// TIA Portal project "SCDW_TEST_67391275" (V17)

(* hardware
DEVICE "SCDW_TEST_PLC"  S7-1200 Station
   slot 0: "Rack_0"  S7-1200 Rack  Rack  V1.0
   slot 1: "SCDW_TEST_PLC"  CPU 1214C AC/DC/Rly  6ES7 214-1BG40-0XB0  V4.4
*)

// ===== PLC "SCDW_TEST_PLC"  CPU 1214C AC/DC/Rly =====

ORGANIZATION_BLOCK "Main"   // OB1, LAD, ProgramCycle
TITLE = "Main Program Sweep (Cycle)"
{ S7_Optimized_Access := 'TRUE' }
VERSION : 0.1
   VAR_INPUT
      Initial_Call : Bool;   // Initial call of this OB
      Remanence : Bool;   // =True, if remanent data are available
   END_VAR
BEGIN

REGION Network 1
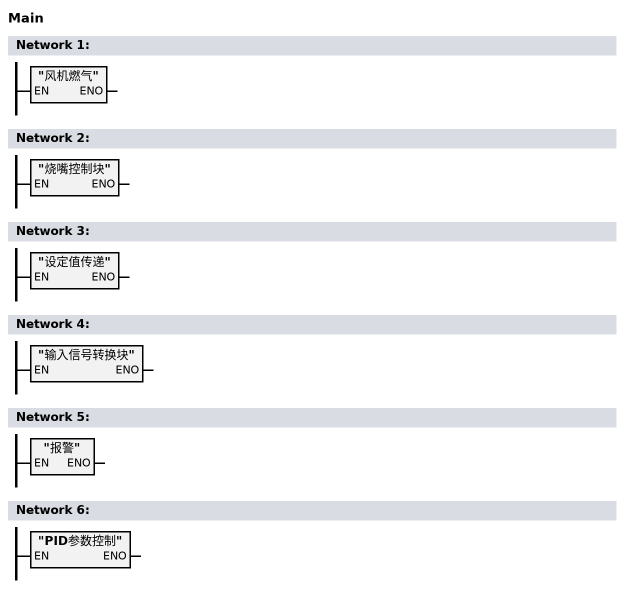
   RUNG wire#powerrail
      "风机燃气"()
   END_RUNG
   // the same network as SCL:
   "风机燃气"();
END_REGION

REGION Network 2
   RUNG wire#powerrail
      "烧嘴控制块"()
   END_RUNG
   // the same network as SCL:
   "烧嘴控制块"();
END_REGION

REGION Network 3
   RUNG wire#powerrail
      "设定值传递"()
   END_RUNG
   // the same network as SCL:
   "设定值传递"();
END_REGION

REGION Network 4
   RUNG wire#powerrail
      "输入信号转换块"()
   END_RUNG
   // the same network as SCL:
   "输入信号转换块"();
END_REGION

REGION Network 5
   RUNG wire#powerrail
      "报警"()
   END_RUNG
   // the same network as SCL:
   "报警"();
END_REGION

REGION Network 6
   RUNG wire#powerrail
      "PID参数控制"()
   END_RUNG
   // the same network as SCL:
   "PID参数控制"();
END_REGION
END_ORGANIZATION_BLOCK